{attribute 'hide_all_locals'}
FUNCTION_BLOCK INTERNAL FB_TimeoutWatcher
VAR_INPUT
    Time_out : TIME := T#0S;
END_VAR
VAR
    IndexOfTaskThatContainsTestSuites : BYTE := 255;
    AdsPort : UINT := TwinCAT_SystemInfoVarList._AppInfo.AdsPort;
    StopCmd : BOOL := FALSE;
    PlcStop : PLC_Stop;
    TimeoutAsULINT : ULINT;
    CpuCounterULINT : ULINT;
    Utility : FB_Utility;
END_VAR

IF Time_out=T#0S OR NOT __ISVALIDREF(GVL_TcUnit.CurrentTestBeingCalled)OR GVL_TcUnit.CurrentTestBeingCalled.TimeStampOfStart=0  THEN
    RETURN;
END_IF

CpuCounterULINT := Utility.GetCpuCounterAsULINT();
TimeOutAsULINT := TIME_TO_ULINT(Time_out) * 10000;
StopCmd := FALSE;

IF IndexOfTaskThatContainsTestSuites = 255 THEN
    IndexOfTaskThatContainsTestSuites := GVL_TcUnit.TestSuiteAddresses[1]^.GetCurrentTaskIndex.index;
END_IF
IF IndexOfTaskThatContainsTestSuites <> 255 THEN
    IF  (CpuCounterULINT >= GVL_TcUnit.CurrentTestBeingCalled.TimeStampOfStart + TimeoutAsULINT) AND NOT GVL_TcUnit.CurrentTestBeingCalled.TestIsFinished THEN
        StopCmd := TRUE;
    END_IF
END_IF
PlcStop(NETID:='',PORT:=AdsPort,STOP:=stopCmd);

END_FUNCTION_BLOCK

(* stored: Version 1.1.0.1, ProductVersion 3.1.4022.18
   POU FB_TimeoutWatcher: Id {c00583a8-41fa-4f83-8876-8a6f8a49c4ec}, SpecialFunc None *)
